// TIA Portal V16 export
// export: Created 2021-04-11T09:51:21.2242374Z, ExportSetting WithDefaults, DisplayName Totally Integrated Automation Portal, DisplayVersion V16, DisplayName TIA Portal Version Control Interface, DisplayVersion V16, DisplayName TIA Portal Openness, DisplayVersion V16, DisplayName STEP 7 Professional, DisplayVersion V16, DisplayName STEP 7 Safety, DisplayVersion V16, DisplayName WinCC Unified SCADA Engineering System, DisplayVersion V16
ORGANIZATION_BLOCK "Main"   // OB1, LAD, ProgramCycle
TITLE = "Main Program Sweep (Cycle)"
{ S7_Optimized_Access := 'TRUE' }
VERSION : 0.1
// stored: AutoNumber true, IsIECCheckEnabled false, SetENOAutomatically false
   VAR_INPUT
      Initial_Call : Bool;   // Initial call of this OB
      Remanence : Bool;   // =True, if remanent data are available
   END_VAR
BEGIN

REGION Network 1: опрос весов
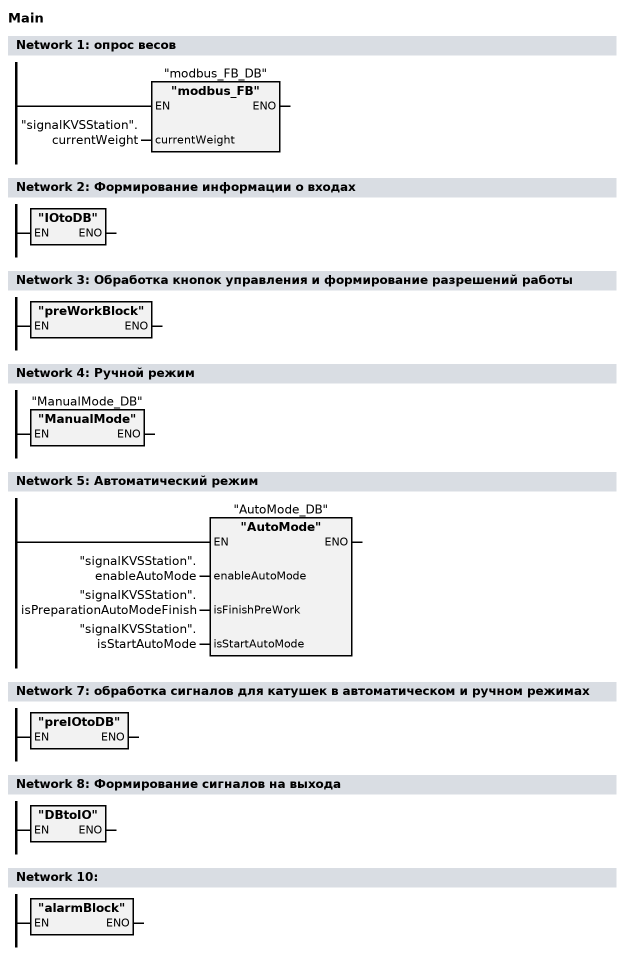
   RUNG wire#powerrail
      "modbus_FB_DB"(currentWeight := "signalKVSStation".currentWeight)
   END_RUNG
   // the same network as SCL:
   "modbus_FB_DB"(currentWeight := "signalKVSStation".currentWeight);   // "modbus_FB"
END_REGION

REGION Network 2: Формирование информации о входах
   RUNG wire#powerrail
      "IOtoDB"()
   END_RUNG
   // the same network as SCL:
   "IOtoDB"();
END_REGION

REGION Network 3: Обработка кнопок управления и формирование разрешений работы
   RUNG wire#powerrail
      "preWorkBlock"()
   END_RUNG
   // the same network as SCL:
   "preWorkBlock"();
END_REGION

REGION Network 4: Ручной режим
   RUNG wire#powerrail
      "ManualMode_DB"()
   END_RUNG
   // the same network as SCL:
   "ManualMode_DB"();   // "ManualMode"
END_REGION

REGION Network 5: Автоматический режим
   RUNG wire#powerrail
      "AutoMode_DB"(enableAutoMode := "signalKVSStation".enableAutoMode, isFinishPreWork := "signalKVSStation".isPreparationAutoModeFinish, isStartAutoMode := "signalKVSStation".isStartAutoMode)
   END_RUNG
   // the same network as SCL:
   "AutoMode_DB"(enableAutoMode := "signalKVSStation".enableAutoMode,   // "AutoMode"
                 isFinishPreWork := "signalKVSStation".isPreparationAutoModeFinish,
                 isStartAutoMode := "signalKVSStation".isStartAutoMode);
END_REGION

REGION Network 7: обработка сигналов для катушек в автоматическом и ручном режимах
   RUNG wire#powerrail
      "preIOtoDB"()
   END_RUNG
   // the same network as SCL:
   "preIOtoDB"();
END_REGION

REGION Network 8: Формирование сигналов на выхода
   RUNG wire#powerrail
      "DBtoIO"()
   END_RUNG
   // the same network as SCL:
   "DBtoIO"();
END_REGION

REGION Network 10
   RUNG wire#powerrail
      "alarmBlock"()
   END_RUNG
   // the same network as SCL:
   "alarmBlock"();
END_REGION
END_ORGANIZATION_BLOCK
